(* IEC 61131-3 sources: AXOpen/src/components.rexroth.tightening/ctrl/src/TemplateComponent (part 3) *)

                IF _progress = 475 THEN                                                                                     // TemplateTask_20steps_6 running: , <add the detailed description of the current action 16>
                    TaskMessenger.ActivateOnCondition(ULINT#675, _infoTimer.output, eAxoMessageCategory#Warning);
                    IF _infoTimer.output THEN
                        Status.Error.Id := UINT#675;
                    END_IF;

                    IF TRUE THEN
                        THIS.CallTimers(FALSE);
                        _progress := 476;
                    END_IF;
                END_IF;

                IF _progress = 476 THEN                                                                                     // TemplateTask_20steps_6 running: , <add the detailed description of the current action 17>
                    TaskMessenger.ActivateOnCondition(ULINT#676, _infoTimer.output, eAxoMessageCategory#Warning);
                    IF _infoTimer.output THEN
                        Status.Error.Id := UINT#676;
                    END_IF;

                    IF TRUE THEN
                        THIS.CallTimers(FALSE);
                        _progress := 477;
                    END_IF;
                END_IF;

                IF _progress = 477 THEN                                                                                     // TemplateTask_20steps_6 running: , <add the detailed description of the current action 18>
                    TaskMessenger.ActivateOnCondition(ULINT#677, _infoTimer.output, eAxoMessageCategory#Warning);
                    IF _infoTimer.output THEN
                        Status.Error.Id := UINT#677;
                    END_IF;

                    IF TRUE THEN
                        THIS.CallTimers(FALSE);
                        _progress := 478;
                    END_IF;
                END_IF;

                IF _progress = 478 THEN                                                                                     // TemplateTask_20steps_6 running: , <add the detailed description of the current action 19>
                    TaskMessenger.ActivateOnCondition(ULINT#678, _infoTimer.output, eAxoMessageCategory#Warning);
                    IF _infoTimer.output THEN
                        Status.Error.Id := UINT#678;
                    END_IF;

                    IF TRUE THEN
                        THIS.CallTimers(FALSE);
                        _progress := 479;
                    END_IF;
                END_IF;

                IF _progress = 479 THEN                                                                                     // TemplateTask_20steps_6 running: , <add the detailed description of the current action 20>
                    TemplateTask_20steps_6.DoneWhen(TRUE);
                END_IF;

                THIS.CallTimers(TRUE);

                TemplateTask_20steps_6.ThrowWhen(_errorTimer.output);
                Status.Action.Id := TO_UINT(_progress);
                TemplateTask_20steps_6.ThrowWhen(TemplateTask_20steps_6.Duration >= Config.ErrorTime ,'TemplateTask_20steps_6 error.');
            END_IF;
            IF TemplateTask_20steps_6.DoneReached() THEN
                Status.Action.Id :=  UINT#261;
                Status.Error.Id :=  UINT#0;
            ELSIF TemplateTask_20steps_6.ErrorOccured() THEN
                Status.Action.Id :=  UINT#1060;
                Status.Error.Id  :=  UINT#1060;
            ELSIF TemplateTask_20steps_6.AbortTriggered()THEN
                Status.Action.Id :=  UINT#1061;
                Status.Error.Id  :=  UINT#1061;
            END_IF;
            Messenger.ActivateOnCondition(ULINT#1060,TemplateTask_20steps_6.HasError(), eAxoMessageCategory#Error);
            Messenger.ActivateOnCondition(ULINT#1061,TemplateTask_20steps_6.IsAborted(), eAxoMessageCategory#Error);
            Messenger.ActivateOnCondition(ULINT#262,TemplateTask_20steps_6.RestoreTriggered() , eAxoMessageCategory#Error);
            IF TemplateTask_20steps_6.RestoreTriggered() AND _progress >= 460 AND _progress <= 479  THEN
                Status.Action.Id :=  UINT#262;
                _progress := 0;
            END_IF;
            //******************************************

            //***********Update outputs ****************
            // _data_out_1[0].%X1                  :=      TemplateComponentOutputStructure_hwID_11.Item1;
            // _data_out_1[0].%X2                  :=      TemplateComponentOutputStructure_hwID_11.Item2;
            // _data_out_1[0].%X3                  :=      TemplateComponentOutputStructure_hwID_11.Item1;
            // _data_out_1[0].%X4                  :=      TemplateComponentOutputStructure_hwID_11.Item2;

            _returnValue := Siemens.Simatic.S71500.DistributedIO.WriteData(_hwID_11,_data_out_1);
            IF _returnValue > WORD#0 THEN
                Messenger.Activate(UINT#871, eAxoMessageCategory#ProgrammingError);
                Status.Error.Id := UINT#871;
                RETURN;
            END_IF;

            // _data_out_1[0].%X1                  :=      TemplateComponentOutputStructure_hwID_12.Item1;
            // _data_out_1[0].%X2                  :=      TemplateComponentOutputStructure_hwID_12.Item2;
            // _data_out_1[0].%X3                  :=      TemplateComponentOutputStructure_hwID_12.Item1;
            // _data_out_1[0].%X4                  :=      TemplateComponentOutputStructure_hwID_12.Item2;

            _returnValue := Siemens.Simatic.S71500.DistributedIO.WriteData(_hwID_12,_data_out_1);
            IF _returnValue > WORD#0 THEN
                Messenger.Activate(UINT#872, eAxoMessageCategory#ProgrammingError);
                Status.Error.Id := UINT#872;
                RETURN;
            END_IF;

            // _data_out_4[1]                     :=      TO_WORD(TemplateComponentOutputStructure_hwID_13.Item1).%B0;
            // _data_out_4[0]                     :=      TO_WORD(TemplateComponentOutputStructure_hwID_13.Item1).%B1;
            // _data_out_4[3]                     :=      TO_WORD(TemplateComponentOutputStructure_hwID_13.Item2).%B0;
            // _data_out_4[2]                     :=      TO_WORD(TemplateComponentOutputStructure_hwID_13.Item2).%B1;

            _returnValue := Siemens.Simatic.S71500.DistributedIO.WriteData(_hwID_13,_data_out_4);
            IF _returnValue > WORD#0 THEN
                Messenger.Activate(UINT#873, eAxoMessageCategory#ProgrammingError);
                Status.Error.Id := UINT#873;
                RETURN;
            END_IF;

            // _data_out_8[3]                     :=      TO_DWORD(TemplateComponentOutputStructure_hwID_14.Item1).%B0;
            // _data_out_8[2]                     :=      TO_DWORD(TemplateComponentOutputStructure_hwID_14.Item1).%B1;
            // _data_out_8[1]                     :=      TO_DWORD(TemplateComponentOutputStructure_hwID_14.Item1).%B2;
            // _data_out_8[0]                     :=      TO_DWORD(TemplateComponentOutputStructure_hwID_14.Item1).%B3;
            // _data_out_8[7]                     :=      TO_DWORD(TemplateComponentOutputStructure_hwID_14.Item2).%B0;
            // _data_out_8[6]                     :=      TO_DWORD(TemplateComponentOutputStructure_hwID_14.Item2).%B1;
            // _data_out_8[5]                     :=      TO_DWORD(TemplateComponentOutputStructure_hwID_14.Item2).%B2;
            // _data_out_8[4]                     :=      TO_DWORD(TemplateComponentOutputStructure_hwID_14.Item2).%B3;

            _returnValue := Siemens.Simatic.S71500.DistributedIO.WriteData(_hwID_14,_data_out_8);
            IF _returnValue > WORD#0 THEN
                Messenger.Activate(UINT#874, eAxoMessageCategory#ProgrammingError);
                Status.Error.Id := UINT#874;
                RETURN;
            END_IF;

            // _data_out_8[3]                     :=      TO_DWORD(TemplateComponentOutputStructure_hwID_15.Item1).%B0;
            // _data_out_8[2]                     :=      TO_DWORD(TemplateComponentOutputStructure_hwID_15.Item1).%B1;
            // _data_out_8[1]                     :=      TO_DWORD(TemplateComponentOutputStructure_hwID_15.Item1).%B2;
            // _data_out_8[0]                     :=      TO_DWORD(TemplateComponentOutputStructure_hwID_15.Item1).%B3;
            // _data_out_8[7]                     :=      TO_DWORD(TemplateComponentOutputStructure_hwID_15.Item2).%B0;
            // _data_out_8[6]                     :=      TO_DWORD(TemplateComponentOutputStructure_hwID_15.Item2).%B1;
            // _data_out_8[5]                     :=      TO_DWORD(TemplateComponentOutputStructure_hwID_15.Item2).%B2;
            // _data_out_8[4]                     :=      TO_DWORD(TemplateComponentOutputStructure_hwID_15.Item2).%B3;

            _returnValue := Siemens.Simatic.S71500.DistributedIO.WriteData(_hwID_15,_data_out_8);
            IF _returnValue > WORD#0 THEN
                Messenger.Activate(UINT#875, eAxoMessageCategory#ProgrammingError);
                Status.Error.Id := UINT#875;
                RETURN;
            END_IF;

            // _data_out_8[3]                     :=      TO_DWORD(TemplateComponentOutputStructure_hwID_16.Item1).%B0;
            // _data_out_8[2]                     :=      TO_DWORD(TemplateComponentOutputStructure_hwID_16.Item1).%B1;
            // _data_out_8[1]                     :=      TO_DWORD(TemplateComponentOutputStructure_hwID_16.Item1).%B2;
            // _data_out_8[0]                     :=      TO_DWORD(TemplateComponentOutputStructure_hwID_16.Item1).%B3;
            // _data_out_8[7]                     :=      TO_DWORD(TemplateComponentOutputStructure_hwID_16.Item2).%B0;
            // _data_out_8[6]                     :=      TO_DWORD(TemplateComponentOutputStructure_hwID_16.Item2).%B1;
            // _data_out_8[5]                     :=      TO_DWORD(TemplateComponentOutputStructure_hwID_16.Item2).%B2;
            // _data_out_8[4]                     :=      TO_DWORD(TemplateComponentOutputStructure_hwID_16.Item2).%B3;

            _returnValue := Siemens.Simatic.S71500.DistributedIO.WriteData(_hwID_16,_data_out_8);
            IF _returnValue > WORD#0 THEN
                Messenger.Activate(UINT#876, eAxoMessageCategory#ProgrammingError);
                Status.Error.Id := UINT#876;
                RETURN;
            END_IF;

            // _data_out_8[3]                     :=      TO_DWORD(TemplateComponentOutputStructure_hwID_17.Item1).%B0;
            // _data_out_8[2]                     :=      TO_DWORD(TemplateComponentOutputStructure_hwID_17.Item1).%B1;
            // _data_out_8[1]                     :=      TO_DWORD(TemplateComponentOutputStructure_hwID_17.Item1).%B2;
            // _data_out_8[0]                     :=      TO_DWORD(TemplateComponentOutputStructure_hwID_17.Item1).%B3;
            // _data_out_8[7]                     :=      TO_DWORD(TemplateComponentOutputStructure_hwID_17.Item2).%B0;
            // _data_out_8[6]                     :=      TO_DWORD(TemplateComponentOutputStructure_hwID_17.Item2).%B1;
            // _data_out_8[5]                     :=      TO_DWORD(TemplateComponentOutputStructure_hwID_17.Item2).%B2;
            // _data_out_8[4]                     :=      TO_DWORD(TemplateComponentOutputStructure_hwID_17.Item2).%B3;

            _returnValue := Siemens.Simatic.S71500.DistributedIO.WriteData(_hwID_17,_data_out_8);
            IF _returnValue > WORD#0 THEN
                Messenger.Activate(UINT#877, eAxoMessageCategory#ProgrammingError);
                Status.Error.Id := UINT#877;
                RETURN;
            END_IF;

            // _data_out_8[3]                     :=      TO_DWORD(TemplateComponentOutputStructure_hwID_18.Item1).%B0;
            // _data_out_8[2]                     :=      TO_DWORD(TemplateComponentOutputStructure_hwID_18.Item1).%B1;
            // _data_out_8[1]                     :=      TO_DWORD(TemplateComponentOutputStructure_hwID_18.Item1).%B2;
            // _data_out_8[0]                     :=      TO_DWORD(TemplateComponentOutputStructure_hwID_18.Item1).%B3;
            // _data_out_8[7]                     :=      TO_DWORD(TemplateComponentOutputStructure_hwID_18.Item2).%B0;
            // _data_out_8[6]                     :=      TO_DWORD(TemplateComponentOutputStructure_hwID_18.Item2).%B1;
            // _data_out_8[5]                     :=      TO_DWORD(TemplateComponentOutputStructure_hwID_18.Item2).%B2;
            // _data_out_8[4]                     :=      TO_DWORD(TemplateComponentOutputStructure_hwID_18.Item2).%B3;

            _returnValue := Siemens.Simatic.S71500.DistributedIO.WriteData(_hwID_18,_data_out_8);
            IF _returnValue > WORD#0 THEN
                Messenger.Activate(UINT#878, eAxoMessageCategory#ProgrammingError);
                Status.Error.Id := UINT#878;
                RETURN;
            END_IF;

            // _data_out_8[3]                     :=      TO_DWORD(TemplateComponentOutputStructure_hwID_19.Item1).%B0;
            // _data_out_8[2]                     :=      TO_DWORD(TemplateComponentOutputStructure_hwID_19.Item1).%B1;
            // _data_out_8[1]                     :=      TO_DWORD(TemplateComponentOutputStructure_hwID_19.Item1).%B2;
            // _data_out_8[0]                     :=      TO_DWORD(TemplateComponentOutputStructure_hwID_19.Item1).%B3;
            // _data_out_8[7]                     :=      TO_DWORD(TemplateComponentOutputStructure_hwID_19.Item2).%B0;
            // _data_out_8[6]                     :=      TO_DWORD(TemplateComponentOutputStructure_hwID_19.Item2).%B1;
            // _data_out_8[5]                     :=      TO_DWORD(TemplateComponentOutputStructure_hwID_19.Item2).%B2;
            // _data_out_8[4]                     :=      TO_DWORD(TemplateComponentOutputStructure_hwID_19.Item2).%B3;

            _returnValue := Siemens.Simatic.S71500.DistributedIO.WriteData(_hwID_19,_data_out_8);
            IF _returnValue > WORD#0 THEN
                Messenger.Activate(UINT#879, eAxoMessageCategory#ProgrammingError);
                Status.Error.Id := UINT#879;
                RETURN;
            END_IF;

            // _data_out_8[3]                     :=      TO_DWORD(TemplateComponentOutputStructure_hwID_20.Item1).%B0;
            // _data_out_8[2]                     :=      TO_DWORD(TemplateComponentOutputStructure_hwID_20.Item1).%B1;
            // _data_out_8[1]                     :=      TO_DWORD(TemplateComponentOutputStructure_hwID_20.Item1).%B2;
            // _data_out_8[0]                     :=      TO_DWORD(TemplateComponentOutputStructure_hwID_20.Item1).%B3;
            // _data_out_8[7]                     :=      TO_DWORD(TemplateComponentOutputStructure_hwID_20.Item2).%B0;
            // _data_out_8[6]                     :=      TO_DWORD(TemplateComponentOutputStructure_hwID_20.Item2).%B1;
            // _data_out_8[5]                     :=      TO_DWORD(TemplateComponentOutputStructure_hwID_20.Item2).%B2;
            // _data_out_8[4]                     :=      TO_DWORD(TemplateComponentOutputStructure_hwID_20.Item2).%B3;

            _returnValue := Siemens.Simatic.S71500.DistributedIO.WriteData(_hwID_20,_data_out_8);
            IF _returnValue > WORD#0 THEN
                Messenger.Activate(UINT#880, eAxoMessageCategory#ProgrammingError);
                Status.Error.Id := UINT#880;
                RETURN;
            END_IF;

            //******************************************

        END_METHOD

        METHOD PUBLIC TemplateMethod_10steps_1 : IAxoTaskState
            TemplateMethod_10steps_1 := TemplateTask_10steps_1.Invoke(THIS);
        END_METHOD

        METHOD PUBLIC TemplateMethod_10steps_2 : IAxoTaskState
            TemplateMethod_10steps_2 := TemplateTask_10steps_2.Invoke(THIS);
        END_METHOD

        METHOD PUBLIC TemplateMethod_10steps_3 : IAxoTaskState
            TemplateMethod_10steps_3 := TemplateTask_10steps_3.Invoke(THIS);
        END_METHOD

        METHOD PUBLIC TemplateMethod_10steps_4 : IAxoTaskState
            TemplateMethod_10steps_4 := TemplateTask_10steps_4.Invoke(THIS);
        END_METHOD

        METHOD PUBLIC TemplateMethod_10steps_5 : IAxoTaskState
            TemplateMethod_10steps_5 := TemplateTask_10steps_5.Invoke(THIS);
        END_METHOD

        METHOD PUBLIC TemplateMethod_10steps_6 : IAxoTaskState
            TemplateMethod_10steps_6 := TemplateTask_10steps_6.Invoke(THIS);
        END_METHOD

        METHOD PUBLIC TemplateMethod_20steps_1 : IAxoTaskState
            TemplateMethod_20steps_1 := TemplateTask_20steps_1.Invoke(THIS);
        END_METHOD

        METHOD PUBLIC TemplateMethod_20steps_2 : IAxoTaskState
            TemplateMethod_20steps_2 := TemplateTask_20steps_2.Invoke(THIS);
        END_METHOD

        METHOD PUBLIC TemplateMethod_20steps_3 : IAxoTaskState
            TemplateMethod_20steps_3 := TemplateTask_20steps_3.Invoke(THIS);
        END_METHOD

        METHOD PUBLIC TemplateMethod_20steps_4 : IAxoTaskState
            TemplateMethod_20steps_4 := TemplateTask_20steps_4.Invoke(THIS);
        END_METHOD

        METHOD PUBLIC TemplateMethod_20steps_5 : IAxoTaskState
            TemplateMethod_20steps_5 := TemplateTask_20steps_5.Invoke(THIS);
        END_METHOD

        METHOD PUBLIC TemplateMethod_20steps_6 : IAxoTaskState
            TemplateMethod_20steps_6 := TemplateTask_20steps_6.Invoke(THIS);
        END_METHOD

        METHOD PROTECTED OVERRIDE ManualControl
            THIS._isManuallyControllable := true;
        END_METHOD

        ///<summary>
        /// Restores this component into intial state.
        ///</summary>
        METHOD PUBLIC OVERRIDE Restore
            VAR
                _index : INT;
            END_VAR
            Status.Action.Id := UINT#0;
            Status.Error.Id  := UINT#0;

            _progress       :=   INT#0;
            _returnValue    :=   WORD#0;

            _data_out_1[0] := BYTE#0;
            _data_out_2[0] := BYTE#0;
            _data_out_2[1] := BYTE#0;

            FOR _index := 0 TO 3 DO
                _data_in[_index] := BYTE#0;
                _data_out_4[_index] := BYTE#0;
                _data_out_8[_index] := BYTE#0;
                _data_out_255[_index] := BYTE#0;
            END_FOR;

            FOR _index := 4 TO 7 DO
                _data_in[_index] := BYTE#0;
                _data_out_8[_index] := BYTE#0;
                _data_out_255[_index] := BYTE#0;
            END_FOR;

            FOR _index := 8 TO 254 DO
                _data_in[_index] := BYTE#0;
                _data_out_255[_index] := BYTE#0;
            END_FOR;

            _word           :=   WORD#0;
            _dword          :=   DWORD#0;

            TemplateTask_10steps_1.Restore();
            TemplateTask_10steps_2.Restore();
            TemplateTask_10steps_3.Restore();
            TemplateTask_10steps_4.Restore();
            TemplateTask_10steps_5.Restore();
            TemplateTask_10steps_6.Restore();
            TemplateTask_20steps_1.Restore();
            TemplateTask_20steps_2.Restore();
            TemplateTask_20steps_3.Restore();
            TemplateTask_20steps_4.Restore();
            TemplateTask_20steps_5.Restore();
            TemplateTask_20steps_6.Restore();
            HardwareDiagnosticsTask.Restore();

            Status.Action.Id := UINT#50;
            RestoreTask.DoneWhen(TRUE);

        END_METHOD

        METHOD PRIVATE CallTimers
            VAR_INPUT
                signal : BOOL;
            END_VAR

            _infoTimer.OnDelay(THIS, signal ,Config.InfoTime);
            _errorTimer.OnDelay(THIS, signal , Config.ErrorTime);
        END_METHOD

    END_CLASS
END_NAMESPACE
